Staubli VAL3: pallet.dtx

mdesc mNomSpeed
public pointRx pO = {fatherId=world[0]}
public pointRx pX = {fatherId=world[0]}
public pointRx pY = {fatherId=world[0]}
public num ndX
public num ndY
public pointRx pStart = {fatherId=world[0]}
public frame fFrame = {fatherId=world[0]}
public string sToolName
